// TIA Portal project "Simple Siemens PLC Ladder Logic Examples to Learn" (V17)
// Simple Siemens PLC Ladder Logic Examples to Learn

(* hardware
DEVICE "S7-1200 station_1"  S7-1200 Station
   slot 0: "Rack_0"  S7-1200 Rack  Rack  V1.0
   slot 1: "PLC_1"  CPU 1211C AC/DC/Rly  6ES7 211-1BE40-0XB0  V4.5
*)

// ===== PLC "PLC_1"  CPU 1211C AC/DC/Rly =====

VAR_GLOBAL   // PLC tag table "Default tag table"
   "A" AT %I0.0 : Bool;
   "B" AT %I0.1 : Bool;
   "C" AT %I0.2 : Bool;
   "D" AT %I0.3 : Bool;
   "E" AT %I0.4 : Bool;
   "Y (Output)" AT %Q0.0 : Bool;
END_VAR

ORGANIZATION_BLOCK "Main"   // OB1, LAD, ProgramCycle
TITLE = "Main Program Sweep (Cycle)"
{ S7_Optimized_Access := 'TRUE' }
VERSION : 0.1
   VAR_INPUT
      Initial_Call : Bool;   // Initial call of this OB
      Remanence : Bool;   // =True, if remanent data are available
   END_VAR
BEGIN

REGION Network 1
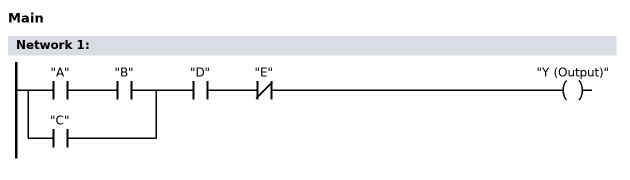
   RUNG wire#powerrail
      Contact( "A" )
      Contact( "B" )
      wire#w1
      Contact( "D" )
      I_Contact( "E" )
      Coil( "Y (Output)" )
   END_RUNG
   RUNG wire#powerrail
      Contact( "C" )
   END_RUNG wire#w1
   // the same network as SCL:
   "Y (Output)" := (("A" AND "B") OR "C") AND "D" AND NOT "E";
END_REGION
END_ORGANIZATION_BLOCK